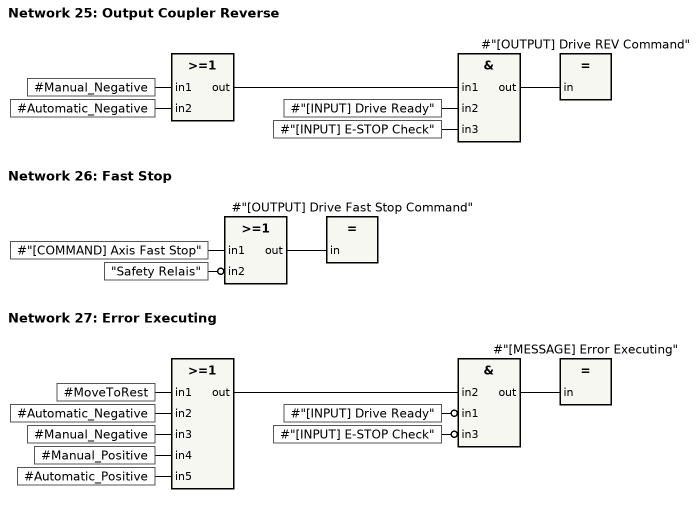
   #"[OUTPUT] Drive REV Command" := (#Manual_Negative OR #Automatic_Negative) AND #"[INPUT] Drive Ready" AND #"[INPUT] E-STOP Check";
END_REGION

REGION Network 26: Fast Stop
   #"[OUTPUT] Drive Fast Stop Command" := #"[COMMAND] Axis Fast Stop" OR NOT "Safety Relais";
END_REGION

REGION Network 27: Error Executing
   #"[MESSAGE] Error Executing" := (#MoveToRest OR #Automatic_Negative OR #Manual_Negative OR #Manual_Positive OR #Automatic_Positive) AND NOT #"[INPUT] Drive Ready" AND NOT #"[INPUT] E-STOP Check";
END_REGION
END_FUNCTION

FUNCTION "EncoderFeedback" : Void   // FC16, FBD
TITLE = EncoderFeedback Block
VERSION : 0.1
// stored: AutoNumber true, IsIECCheckEnabled false, UDAEnableTagReadback false
   VAR_INPUT
      CounterTag : Int;   // Connect to the CounterTag IW102
      Position_Offset : Real;   // Fill in the tolerance, when the axis approves the position. Above or below the desired position
      Pulsfactor : Real;   // Number of pulses after 360 degree turn of the axis.
      Position_Correction : Real;   // Small Position Correction for the Axis
      ReferenceRun_Command : Bool;   // Command of starting the referencerun
      ReferenceSwitch : Bool;   // ReferenceSwitch Mounted on Axis
      ReferencePosition : Int;   // Position where the index puls of the reference switch enters.
   END_VAR
   VAR_OUTPUT
      Scaled_Position : Real;   // Scaled Position scaled with Pulsfactor
      Actual_Enc_Pos : Real;   // Actual Encoder Position
      AxisDB_Connection : Real;   // Connection with Axis DB connection
   END_VAR
   VAR_TEMP
      Corrected_Axis_Pos : Real;
      Unscaled_Position : Int;   // Unscaled Position of the Encoder
      Unsc2 : Int;   // Unsc 2 position
      Act_Enc_Pos_Int : DInt;
      Scaled_Position_Real : Real;
      PosDint : DInt;
      Unscaled_Position_Real : Real;
      InternalCounter : Int;
      CalDifCounter : Int;
      Pos_Storage : Int;
      Pos_Diffrence : Int;
      Add_Pos : Int;
      Sub_Pos : Int;
      LessThanZero : Bool;
      LTZ_out : Int;
   END_VAR
BEGIN

REGION Network 1: SPARE
END_REGION

NETWORK
TITLE = Call the Countermodule
      L     #CounterTag;  //Van tellerkaart TAG Gelinkt aan IW102
      L     "PositionManagement".Data.CntPlsPrev;  //Vorige scan
      -D;
      T     "PositionManagement".Data.CntPlsDiff;  //Verschil

      L     "PositionManagement".Data.CntPlsDiff;  // Verschil groter dan nul?
      L     0;
      >D;
      JCN   chkneg;

      L     "PositionManagement".Data.CntPlsDiff;  //Verschil optellen bij actuele pulswaarde
      L     "PositionManagement".Data.CntPlsAct;
      +D;
      T     "PositionManagement".Data.CntPlsAct;
      JU    end;  //rest overslaan.

chkneg:L     "PositionManagement".Data.CntPlsDiff;  // Verschil groter dan nul?
      L     0;
      <D;
      JCN   end;
      L     -1;  //verschil positief maken
      *D;
      T     "PositionManagement".Data.CntPlsDiff;  //verschil positief

      L     "PositionManagement".Data.CntPlsAct;  //Verschil optellen bij actuele pulswaarde
      +D;
      T     "PositionManagement".Data.CntPlsAct;

end:  NOP   0;

      L     #CounterTag;
      T     "PositionManagement".Data.CntPlsPrev;


REGION Network 3: Store Old Position
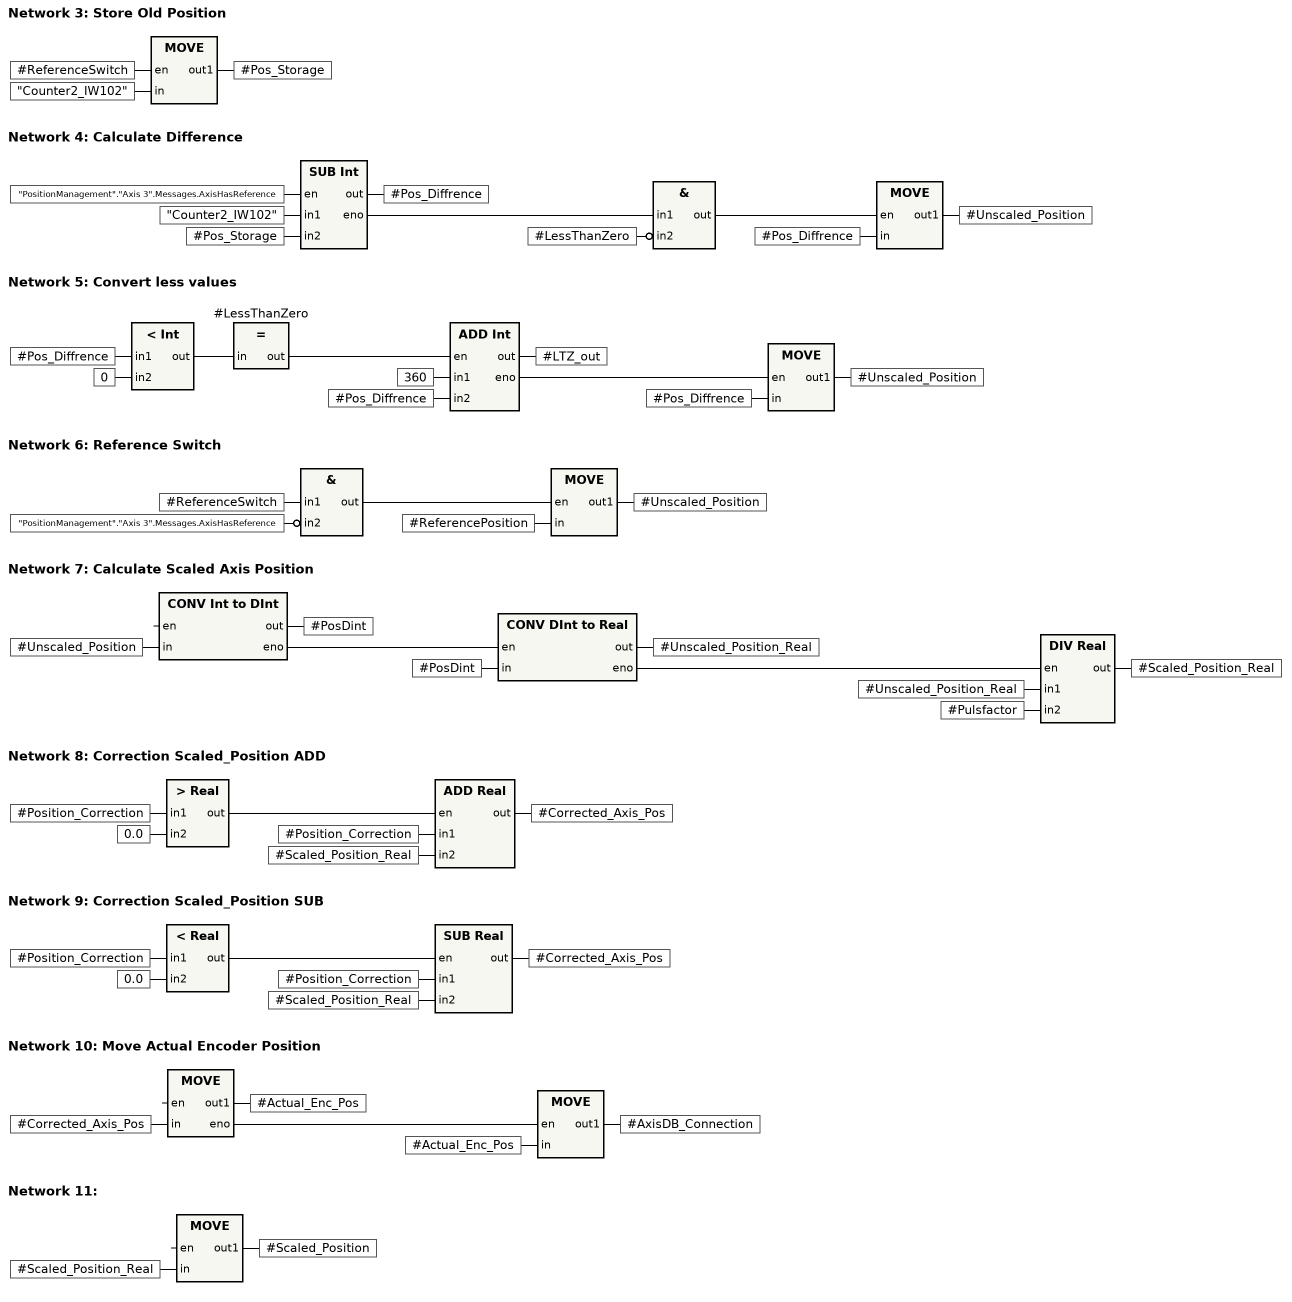
   IF #ReferenceSwitch THEN #Pos_Storage := "Counter2_IW102"; END_IF;
END_REGION

REGION Network 4: Calculate Difference
   // ENO of a box is taken as its EN; it also drops when the box reports an error
   IF "PositionManagement"."Axis 3".Messages.AxisHasReference THEN
       #Pos_Diffrence := "Counter2_IW102" - #Pos_Storage;
   END_IF;
   IF "PositionManagement"."Axis 3".Messages.AxisHasReference AND NOT #LessThanZero THEN
       #Unscaled_Position := #Pos_Diffrence;
   END_IF;
END_REGION

REGION Network 5: Convert less values
   // ENO of a box is taken as its EN; it also drops when the box reports an error
   #LessThanZero := #Pos_Diffrence < 0;
   IF #LessThanZero THEN
       #LTZ_out := 360 + #Pos_Diffrence;
       #Unscaled_Position := #Pos_Diffrence;
   END_IF;
END_REGION

REGION Network 6: Reference Switch
   IF #ReferenceSwitch AND NOT "PositionManagement"."Axis 3".Messages.AxisHasReference THEN
       #Unscaled_Position := #ReferencePosition;
   END_IF;
END_REGION

REGION Network 7: Calculate Scaled Axis Position
   // ENO of a box is taken as its EN; it also drops when the box reports an error
   #PosDint := INT_TO_DINT(#Unscaled_Position);
   #Unscaled_Position_Real := DINT_TO_REAL(#PosDint);
   #Scaled_Position_Real := #Unscaled_Position_Real / #Pulsfactor;
END_REGION

REGION Network 8: Correction Scaled_Position ADD
   IF #Position_Correction > 0.0 THEN
       #Corrected_Axis_Pos := #Position_Correction + #Scaled_Position_Real;
   END_IF;
END_REGION

REGION Network 9: Correction Scaled_Position SUB
   IF #Position_Correction < 0.0 THEN
       #Corrected_Axis_Pos := #Position_Correction - #Scaled_Position_Real;
   END_IF;
END_REGION

REGION Network 10: Move Actual Encoder Position
   // ENO of a box is taken as its EN; it also drops when the box reports an error
   #Actual_Enc_Pos := #Corrected_Axis_Pos;
   #AxisDB_Connection := #Actual_Enc_Pos;
END_REGION

REGION Network 11
   #Scaled_Position := #Scaled_Position_Real;
END_REGION
END_FUNCTION

FUNCTION_BLOCK "MC_Move"   // FB10, FBD
TITLE = MC_Move
VERSION : 0.1
// Block moves an Axis to an Desired Position, this block comes with the brake feature. When the axis is on position it keeps the brake for a time. You can set the time in the Brake Time field.
// stored: AutoNumber true, IsIECCheckEnabled false, UDAEnableTagReadback false
   VAR_INPUT
      Start : Bool;
      "Desired Position" : Real;
      "Speed (50-75%)" : Int;
      "Brake on Position" : Bool;
      Acceleration : Real;
      Deacceleration : Real;
      "Drive Ready" : Bool;
      "Drive On Position" : Bool;
      "Brake Time" : Time := T#500ms;
      "Safety OK" : Bool;
   END_VAR
   VAR_OUTPUT
      Go : Bool;
      "Desired Position Out" : Real;
      "Speed Output" : Int;
      "Acceleration Out" : Real;
      "Deacceleration Out" : Real;
      "Brake Out" : Bool;
   END_VAR
   VAR_TEMP
      SR_1 : Bool;
   END_VAR
BEGIN

REGION Network 1: Start - Go To Position + Speed
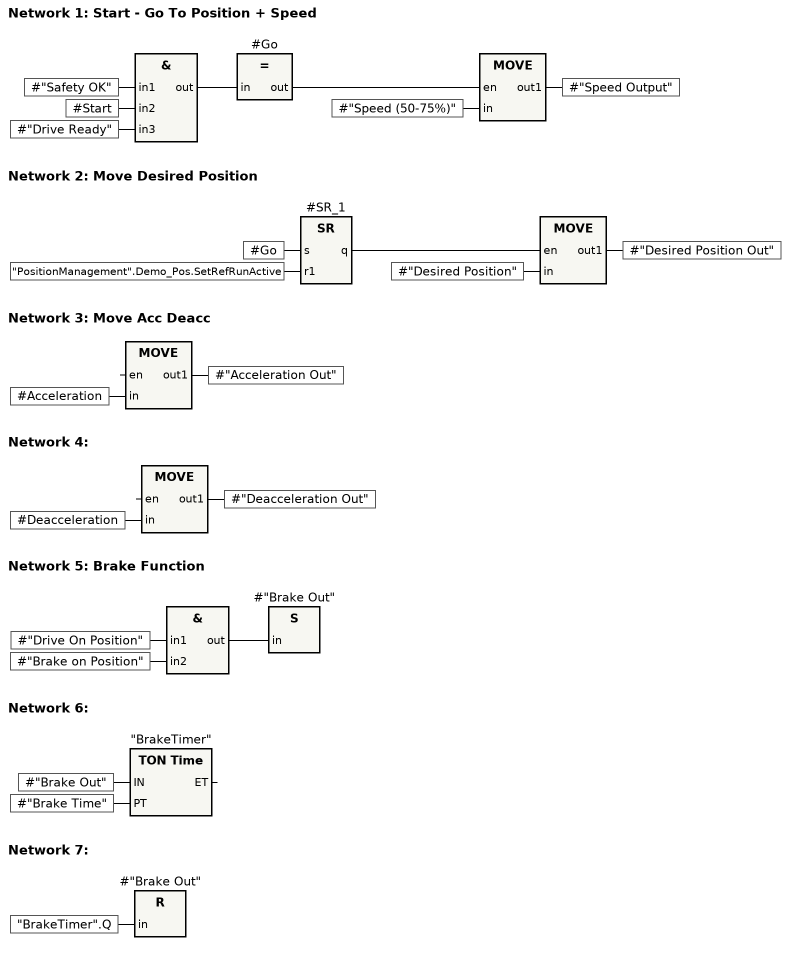
   #Go := #"Safety OK" AND #Start AND #"Drive Ready";
   IF #Go THEN #"Speed Output" := #"Speed (50-75%)"; END_IF;
END_REGION

REGION Network 2: Move Desired Position
   IF #Go THEN
       #SR_1 := TRUE;   // SR flip-flop
   END_IF;
   IF "PositionManagement".Demo_Pos.SetRefRunActive THEN #SR_1 := FALSE; END_IF;
   IF #SR_1 THEN #"Desired Position Out" := #"Desired Position"; END_IF;
END_REGION

REGION Network 3: Move Acc Deacc
   #"Acceleration Out" := #Acceleration;
END_REGION

REGION Network 4
   #"Deacceleration Out" := #Deacceleration;
END_REGION

REGION Network 5: Brake Function
   IF #"Drive On Position" AND #"Brake on Position" THEN #"Brake Out" := TRUE; END_IF;
END_REGION

REGION Network 6
   "BrakeTimer".TON(IN := #"Brake Out", PT := #"Brake Time");
END_REGION

REGION Network 7
   IF "BrakeTimer".Q THEN #"Brake Out" := FALSE; END_IF;
END_REGION
END_FUNCTION_BLOCK

FUNCTION_BLOCK "MC_Jog"   // FB11, FBD
TITLE = MC_Jog
VERSION : 0.1
// With this block you can Jog an Axis manual, you can set the speed on 25%, 50% or 75%. It also has an brake functionality, when you set Brake to true, it holds the brake for 2 seconds, then releases it.
// stored: AutoNumber true, IsIECCheckEnabled false, UDAEnableTagReadback false
   VAR_INPUT
      "Jog Forward" : Bool;
      "Jog Backward" : Bool;
      Speed : Int;
      Brake : Bool;
   END_VAR
   VAR_OUTPUT
      "Drive Fwd Output" : Bool;
      "Drive Rev Output" : Bool;
      "Drive Speed Output" : Int;
      "Drive Brake Output" : Bool;
   END_VAR
BEGIN

REGION Network 1: Manual Control
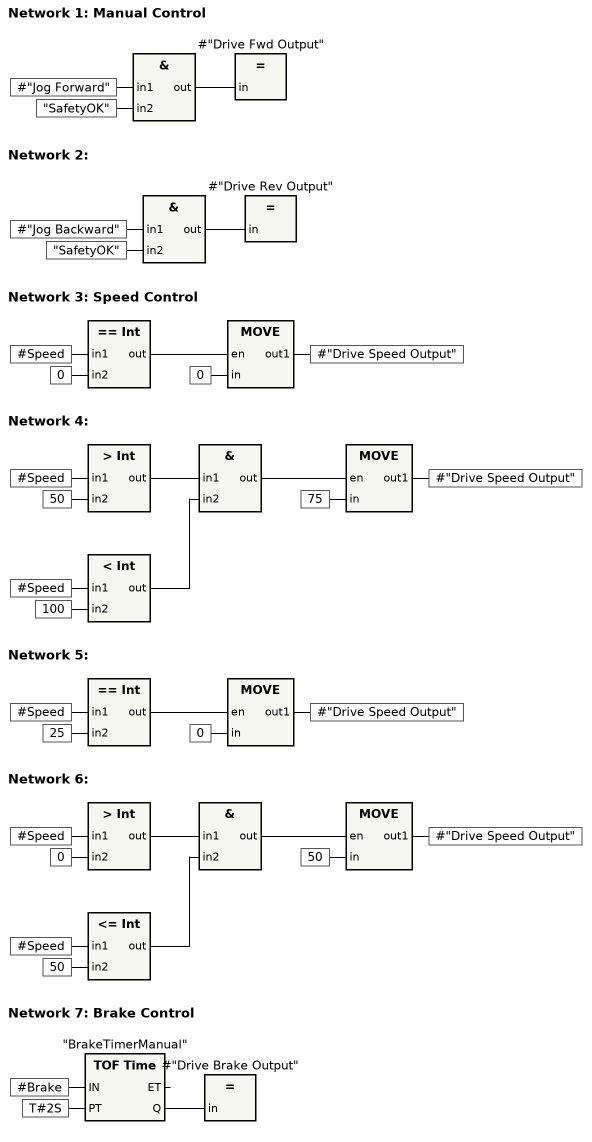
   #"Drive Fwd Output" := #"Jog Forward" AND "SafetyOK";
END_REGION

REGION Network 2
   #"Drive Rev Output" := #"Jog Backward" AND "SafetyOK";
END_REGION

REGION Network 3: Speed Control
   IF #Speed = 0 THEN #"Drive Speed Output" := 0; END_IF;
END_REGION

REGION Network 4
   IF (#Speed > 50) AND (#Speed < 100) THEN #"Drive Speed Output" := 75; END_IF;
END_REGION

REGION Network 5
   IF #Speed = 25 THEN #"Drive Speed Output" := 0; END_IF;
END_REGION

REGION Network 6
   IF (#Speed > 0) AND (#Speed <= 50) THEN #"Drive Speed Output" := 50; END_IF;
END_REGION

REGION Network 7: Brake Control
   "BrakeTimerManual".TOF(IN := #Brake, PT := T#2S);
   #"Drive Brake Output" := "BrakeTimerManual".Q;
END_REGION
END_FUNCTION_BLOCK

FUNCTION_BLOCK "ProductBuffer_V3"
{ S7_Optimized_Access := 'FALSE' }
VERSION : 0.1
   VAR_INPUT 
      SensorInput : Bool;   // Sensor aan begin band
      EncoderPosition : Real;   // Koppel aan Encoder Data Instance
      TriggerDistance : Real;   // Gewenste Afstand Product voor trigger
      TriggerFeedback : Bool;
   END_VAR

   VAR_OUTPUT 
      TriggerMovement : Bool;   // Trigger Start Movement
      ProductCount : Int;   // Count products in buffer
   END_VAR

   VAR 
      ProductBuffer { S7_SetPoint := 'False'} : Array[0..9] of "ProductTrack";
      PrevSensor { S7_SetPoint := 'True'} : Bool;
      MovementActive : Bool;
      i : Int;
      Distance : Real;
   END_VAR


BEGIN
	// 1️⃣ Flankdetectie - detecteer nieuw product
	IF #SensorInput AND NOT #PrevSensor THEN
	    FOR #i := 0 TO 9 DO
	        IF NOT #ProductBuffer[#i].Active THEN
	            #ProductBuffer[#i].StartPosition := #EncoderPosition;
	            #ProductBuffer[#i].Active := TRUE;
	            EXIT;
	        END_IF;
	    END_FOR;
	END_IF;
	#PrevSensor := #SensorInput;
	
	// 2️⃣ Tel actieve producten
	#ProductCount := 0;
	FOR #i := 0 TO 9 DO
	    IF #ProductBuffer[#i].Active THEN
	        #ProductCount := #ProductCount + 1;
	    END_IF;
	END_FOR;
	
	// 3️⃣ Zoek eerste product dat zijn afstand heeft afgelegd
	IF NOT #MovementActive THEN
	    FOR #i := 0 TO 9 DO
	        IF #ProductBuffer[#i].Active THEN
	            #Distance := #EncoderPosition - #ProductBuffer[#i].StartPosition;
	            
	            IF #Distance >= #TriggerDistance THEN
	                #TriggerMovement := TRUE;
	                #MovementActive := TRUE;
	                #ProductBuffer[#i].Active := FALSE;
	                EXIT;
	            END_IF;
	        END_IF;
	    END_FOR;
	END_IF;
	
	// 4️⃣ Wacht op feedback om beweging af te ronden
	IF #MovementActive AND #TriggerFeedback THEN
	    #TriggerMovement := FALSE;
	    #MovementActive := FALSE;
	END_IF;
	
END_FUNCTION_BLOCK

FUNCTION_BLOCK "Programma 1 - Test"   // FB12, GRAPH
VERSION : 0.1
// stored: AcknowledgeErrorsRequired true, AutoNumber true, CreateMinimizedDB false, IsIECCheckEnabled false, LanguageInNetworks LAD, LockOperatingMode false, PermanentILProcessingInMANMode false, SkipSteps false, UDAEnableTagReadback false, WithAlarmHandling true
   VAR_INPUT
      OFF_SQ { ExternalAccessible := 'False'; ExternalVisible := 'False'; ExternalWritable := 'False'} : Bool := false;   // Turn sequence off
      INIT_SQ { ExternalAccessible := 'False'; ExternalVisible := 'False'; ExternalWritable := 'False'} : Bool := false;   // Set sequence to initial state
      ACK_EF { ExternalAccessible := 'False'; ExternalVisible := 'False'; ExternalWritable := 'False'} : Bool := false;   // Acknowledge all errors and faults
      S_PREV { ExternalAccessible := 'False'; ExternalVisible := 'False'; ExternalWritable := 'False'} : Bool := false;   // Output previous step in parameter S_NO
      S_NEXT { ExternalAccessible := 'False'; ExternalVisible := 'False'; ExternalWritable := 'False'} : Bool := false;   // Indicate next step in parameter S_NO
      SW_AUTO { ExternalAccessible := 'False'; ExternalVisible := 'False'; ExternalWritable := 'False'} : Bool := false;   // Automatic mode
      SW_TAP { ExternalAccessible := 'False'; ExternalVisible := 'False'; ExternalWritable := 'False'} : Bool := false;   // Semiautomatic/switch with transition
      SW_TOP { ExternalAccessible := 'False'; ExternalVisible := 'False'; ExternalWritable := 'False'} : Bool := false;   // Semiautomatic/ignore transition
      SW_MAN { ExternalAccessible := 'False'; ExternalVisible := 'False'; ExternalWritable := 'False'} : Bool := false;   // Manual mode
      S_SEL { ExternalAccessible := 'False'; ExternalVisible := 'False'; ExternalWritable := 'False'} : Int := 0;   // Select step to be output to S_NO
      S_ON { ExternalAccessible := 'False'; ExternalVisible := 'False'; ExternalWritable := 'False'} : Bool := false;   // Activate step indicated in S_NO
      S_OFF { ExternalAccessible := 'False'; ExternalVisible := 'False'; ExternalWritable := 'False'} : Bool := false;   // Deactivate step indicated S_NO
      T_PUSH { ExternalAccessible := 'False'; ExternalVisible := 'False'; ExternalWritable := 'False'} : Bool := false;   // Enable transition to switch in semi automatic mode
      "Confimation Position 1" : Bool;
      "Confirmation Position 2" : Bool;
      "Products more than zero" : Bool;
      "Products zero" : Bool;
      "Timer 1" : Time;
   END_VAR
   VAR_OUTPUT
      S_NO { ExternalAccessible := 'False'; ExternalVisible := 'False'; ExternalWritable := 'False'} : Int := 0;   // Step number
      S_MORE { ExternalAccessible := 'False'; ExternalVisible := 'False'; ExternalWritable := 'False'} : Bool := false;   // More steps are available and can be shown in S_NO
      S_ACTIVE { ExternalAccessible := 'False'; ExternalVisible := 'False'; ExternalWritable := 'False'} : Bool := false;   // Step indicated in S_NO is active
      ERR_FLT { ExternalAccessible := 'False'; ExternalVisible := 'False'; ExternalWritable := 'False'} : Bool := false;   // Interlock or supervision group error
      AUTO_ON { ExternalAccessible := 'False'; ExternalVisible := 'False'; ExternalWritable := 'False'} : Bool := false;   // Automatic mode is active
      TAP_ON { ExternalAccessible := 'False'; ExternalVisible := 'False'; ExternalWritable := 'False'} : Bool := false;   // Semiautomatic mode/step with transition enabled
      TOP_ON { ExternalAccessible := 'False'; ExternalVisible := 'False'; ExternalWritable := 'False'} : Bool := false;   // Semiautomatic mode/ignore transition enabled
      MAN_ON { ExternalAccessible := 'False'; ExternalVisible := 'False'; ExternalWritable := 'False'} : Bool := false;   // Manual mode is active
      "Move Position 1" : Bool;
      "Move Position 2" : Bool;
   END_VAR
   VAR DB_SPECIFIC
      S_DISPLAY { ExternalAccessible := 'False'; ExternalVisible := 'False'; ExternalWritable := 'False'} : Int;   // Internal display of output parameter S_NO
      S_SEL_OLD { ExternalAccessible := 'False'; ExternalVisible := 'False'; ExternalWritable := 'False'} : Int;   // Previous value in S_SEL
      S_DISPIDX { ExternalAccessible := 'False'; ExternalVisible := 'False'; ExternalWritable := 'False'} : Byte;   // Index of the step in S_NO
      T_DISPIDX { ExternalAccessible := 'False'; ExternalVisible := 'False'; ExternalWritable := 'False'} : Byte;   // Index of the transition displayed in T_NO
      MOP { ExternalAccessible := 'False'; ExternalVisible := 'False'; ExternalWritable := 'False'} : Struct   // Mode
         AUTO { ExternalAccessible := 'False'; ExternalVisible := 'False'; ExternalWritable := 'False'} : Bool := true;   // Status: automatic mode
         MAN { ExternalAccessible := 'False'; ExternalVisible := 'False'; ExternalWritable := 'False'} : Bool := false;   // Status: manual mode
         TAP { ExternalAccessible := 'False'; ExternalVisible := 'False'; ExternalWritable := 'False'} : Bool := false;   // Status: semi automatic/switch with transition
         TOP { ExternalAccessible := 'False'; ExternalVisible := 'False'; ExternalWritable := 'False'} : Bool := false;   // Status: semi automatic/ignore transition
         ACK_S { ExternalAccessible := 'False'; ExternalVisible := 'False'; ExternalWritable := 'False'} : Bool := false;   // Request: acknowledge step at parameter S_NO
         REG_S { ExternalAccessible := 'False'; ExternalVisible := 'False'; ExternalWritable := 'False'} : Bool := false;   // Request: register step indicated in S_NO
         T_PREV { ExternalAccessible := 'False'; ExternalVisible := 'False'; ExternalWritable := 'False'} : Bool := false;   // Request: output previous valid transition in T_NO
         T_NEXT { ExternalAccessible := 'False'; ExternalVisible := 'False'; ExternalWritable := 'False'} : Bool := false;   // Request: output next valid transition in T_NO
         LOCK { ExternalAccessible := 'False'; ExternalVisible := 'False'; ExternalWritable := 'False'} : Bool := true;   // Status: interlocks activated
         SUP { ExternalAccessible := 'False'; ExternalVisible := 'False'; ExternalWritable := 'False'} : Bool := true;   // Status: supervisions activated
         ACKREQ { ExternalAccessible := 'False'; ExternalVisible := 'False'; ExternalWritable := 'False'} : Bool := true;   // Status: acknowledgment required
         SSKIP { ExternalAccessible := 'False'; ExternalVisible := 'False'; ExternalWritable := 'False'} : Bool := false;   // Status: "Skip steps" enabled
         OFF { ExternalAccessible := 'False'; ExternalVisible := 'False'; ExternalWritable := 'False'} : Bool := false;   // Request: deactivate all steps
         INIT { ExternalAccessible := 'False'; ExternalVisible := 'False'; ExternalWritable := 'False'} : Bool := true;   // Request: set sequence to initial state
         HALT { ExternalAccessible := 'False'; ExternalVisible := 'False'; ExternalWritable := 'False'} : Bool := false;   // Status: sequence halted
         TMS_HALT { ExternalAccessible := 'False'; ExternalVisible := 'False'; ExternalWritable := 'False'} : Bool := false;   // Status: all internal timers held
         OPS_ZERO { ExternalAccessible := 'False'; ExternalVisible := 'False'; ExternalWritable := 'False'} : Bool := false;   // Status: set all operands processed with N, L, D instructions to 0
         SACT_DISP { ExternalAccessible := 'False'; ExternalVisible := 'False'; ExternalWritable := 'False'} : Bool := true;   // Status: display active steps only
         SEF_DISP { ExternalAccessible := 'False'; ExternalVisible := 'False'; ExternalWritable := 'False'} : Bool := false;   // Status: display only steps with errors and disrupted steps
         SALL_DISP { ExternalAccessible := 'False'; ExternalVisible := 'False'; ExternalWritable := 'False'} : Bool := false;   // Status: display all steps
         S_PREV { ExternalAccessible := 'False'; ExternalVisible := 'False'; ExternalWritable := 'False'} : Bool := false;   // Request: output previous step to S_NO
         S_NEXT { ExternalAccessible := 'False'; ExternalVisible := 'False'; ExternalWritable := 'False'} : Bool := false;   // Request: Output next step at S_NO parameter
         S_SELOK { ExternalAccessible := 'False'; ExternalVisible := 'False'; ExternalWritable := 'False'} : Bool := false;   // Request: output step number from S_SEL to S_NO
         S_ON { ExternalAccessible := 'False'; ExternalVisible := 'False'; ExternalWritable := 'False'} : Bool := false;   // Request: activate step indicated in S_NO
         S_OFF { ExternalAccessible := 'False'; ExternalVisible := 'False'; ExternalWritable := 'False'} : Bool := false;   // Request: deactivate step at parameter S_NO
         T_PUSH { ExternalAccessible := 'False'; ExternalVisible := 'False'; ExternalWritable := 'False'} : Bool := false;   // Request: transition switching enabled
         REG { ExternalAccessible := 'False'; ExternalVisible := 'False'; ExternalWritable := 'False'} : Bool := false;   // Request: register all interlock and supervision errors
         ACK { ExternalAccessible := 'False'; ExternalVisible := 'False'; ExternalWritable := 'False'} : Bool := false;   // Request: acknowledge all interlock and supervision errors
         IL_PERM { ExternalAccessible := 'False'; ExternalVisible := 'False'; ExternalWritable := 'False'} : Bool := false;   // Status: permanent processing of all interlocks
         T_PERM { ExternalAccessible := 'False'; ExternalVisible := 'False'; ExternalWritable := 'False'} : Bool := false;   // Status: permanent processing of all transitions
         ILP_MAN { ExternalAccessible := 'False'; ExternalVisible := 'False'; ExternalWritable := 'False'} : Bool := false;   // Status: permanent processing of all interlocks in manual mode
      END_STRUCT;
      TICKS { ExternalAccessible := 'False'; ExternalVisible := 'False'; ExternalWritable := 'False'} : Struct   // Clock speeds
         DELTA { ExternalAccessible := 'False'; ExternalVisible := 'False'; ExternalWritable := 'False'} : Time := T#0ms;   // Time difference between cycles
         OLD { ExternalAccessible := 'False'; ExternalVisible := 'False'; ExternalWritable := 'False'} : Time := T#0ms;   // 10 ms clock counter value in last cycle
         NEW { ExternalAccessible := 'False'; ExternalVisible := 'False'; ExternalWritable := 'False'} : Time := T#0ms;   // 10 ms clock counter value in this cycle
      END_STRUCT;
      SQ_FLAGS { ExternalAccessible := 'False'; ExternalVisible := 'False'; ExternalWritable := 'False'} : Struct   // Sequence bit memory
         ERR_FLT { ExternalAccessible := 'False'; ExternalVisible := 'False'; ExternalWritable := 'False'} : Bool := false;   // Interlock and supervision group error
         ERROR { ExternalAccessible := 'False'; ExternalVisible := 'False'; ExternalWritable := 'False'} : Bool := false;   // Interlock group error
         FAULT { ExternalAccessible := 'False'; ExternalVisible := 'False'; ExternalWritable := 'False'} : Bool := false;   // Supervision group error
         RT_FAIL { ExternalAccessible := 'False'; ExternalVisible := 'False'; ExternalWritable := 'False'} : Bool := false;   // Runtime error
         NO_SNO { ExternalAccessible := 'False'; ExternalVisible := 'False'; ExternalWritable := 'False'} : Bool := false;   // Requested step number not found
         NF_OFL { ExternalAccessible := 'False'; ExternalVisible := 'False'; ExternalWritable := 'False'} : Bool := false;   // Overflow: too many ON or OFF requests
         SA_OFL { ExternalAccessible := 'False'; ExternalVisible := 'False'; ExternalWritable := 'False'} : Bool := false;   // Overflow: too many steps active
         TV_OFL { ExternalAccessible := 'False'; ExternalVisible := 'False'; ExternalWritable := 'False'} : Bool := false;   // Overflow: too many valid transitions
         MSG_OFL { ExternalAccessible := 'False'; ExternalVisible := 'False'; ExternalWritable := 'False'} : Bool := false;   // Overflow: not enough system resources for ALARM_S
         NO_SWI { ExternalAccessible := 'False'; ExternalVisible := 'False'; ExternalWritable := 'False'} : Bool := false;   // Do not switch in this cycle
         CYC_OP { ExternalAccessible := 'False'; ExternalVisible := 'False'; ExternalWritable := 'False'} : Bool := false;   // Cyclic execution of the sequence after initialization
         AS_MSG { ExternalAccessible := 'False'; ExternalVisible := 'False'; ExternalWritable := 'False'} : Bool := true;   // Alarms during runtime enabled or disabled by instruction
         AS_SEND { ExternalAccessible := 'False'; ExternalVisible := 'False'; ExternalWritable := 'False'} : Bool := false;   // Send alarms from WR_USMSG or only enter in diagnostics buffer
         SQ_BUSY { ExternalAccessible := 'False'; ExternalVisible := 'False'; ExternalWritable := 'False'} : Bool := false;   // Internal edge memory bit for sequence processing
         SA_BUSY { ExternalAccessible := 'False'; ExternalVisible := 'False'; ExternalWritable := 'False'} : Bool := false;   // Internal edge memory bit for sequence processing
         AS_SIG { ExternalAccessible := 'False'; ExternalVisible := 'False'; ExternalWritable := 'False'} : Bool := false;   // Edge memory bit for alarms from Alarm_S and Alarm_SQ
      END_STRUCT;
   END_VAR
BEGIN
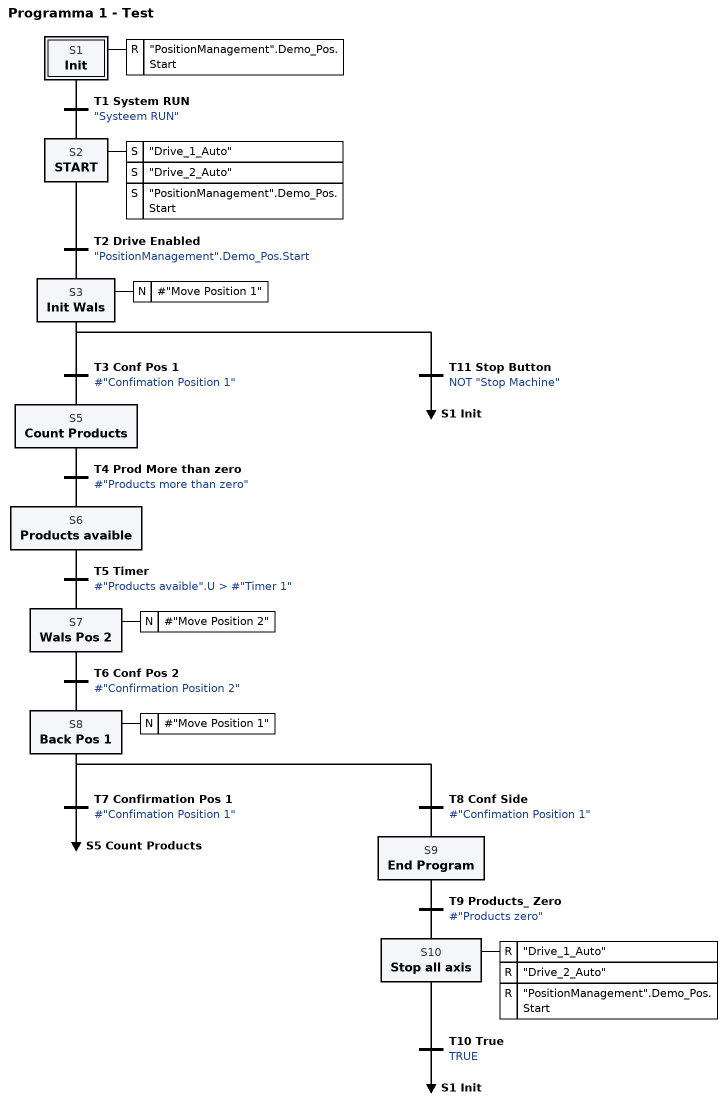
   // sequencer 1: SFC Program
   INITIAL_STEP Init:   // S1
              R    "PositionManagement".Demo_Pos.Start
   END_STEP
   TRANSITION "System RUN" FROM Init TO START   // T1
      := "Systeem RUN";
   END_TRANSITION
   STEP START:   // S2
      // Set Ouputs
              S    "Drive_1_Auto"
              S    "Drive_2_Auto"
              S    "PositionManagement".Demo_Pos.Start
   END_STEP
   TRANSITION "Drive Enabled" FROM START TO "Init Wals"   // T2
      := "PositionManagement".Demo_Pos.Start;
   END_TRANSITION
   STEP "Init Wals":   // S3
      // Move Start Position4
              N    #"Move Position 1"
   END_STEP
   TRANSITION "Conf Pos 1" FROM "Init Wals" TO "Count Products"   // T3
      := #"Confimation Position 1";
   END_TRANSITION
   TRANSITION "Stop Button" FROM "Init Wals" TO Init   // T11, jump
      := NOT "Stop Machine";
   END_TRANSITION
   STEP "Count Products":   // S5
   END_STEP
   TRANSITION "Prod More than zero" FROM "Count Products" TO "Products avaible"   // T4
      := #"Products more than zero";
   END_TRANSITION
   STEP "Products avaible":   // S6
   END_STEP
   TRANSITION "Timer" FROM "Products avaible" TO "Wals Pos 2"   // T5: Timer 1
      := #"Products avaible".U > #"Timer 1";
   END_TRANSITION
   STEP "Wals Pos 2":   // S7
              N    #"Move Position 2"
   END_STEP
   TRANSITION "Conf Pos 2" FROM "Wals Pos 2" TO "Back Pos 1"   // T6
      := #"Confirmation Position 2";
   END_TRANSITION
   STEP "Back Pos 1":   // S8
      // Move Position 1
              N    #"Move Position 1"
   END_STEP
   TRANSITION "Confirmation Pos 1" FROM "Back Pos 1" TO "Count Products"   // T7, jump: Conf Pos 1
      := #"Confimation Position 1";
   END_TRANSITION
   TRANSITION "Conf Side" FROM "Back Pos 1" TO "End Program"   // T8
      := #"Confimation Position 1";
   END_TRANSITION
   STEP "End Program":   // S9
   END_STEP
   TRANSITION "Products_ Zero" FROM "End Program" TO "Stop all axis"   // T9
      := #"Products zero";
   END_TRANSITION
   STEP "Stop all axis":   // S10
      // Reset Axis
              R    "Drive_1_Auto"
              R    "Drive_2_Auto"
              R    "PositionManagement".Demo_Pos.Start
   END_STEP
   TRANSITION True FROM "Stop all axis" TO Init   // T10, jump
      := TRUE;
   END_TRANSITION
END_FUNCTION_BLOCK

FUNCTION_BLOCK "Ouput_Function_1"   // FB8, FBD
TITLE = Ouput Controller Function Block
VERSION : 0.1
// stored: AutoNumber true, IsIECCheckEnabled false, UDAEnableTagReadback false
   VAR_INPUT
      "Stop Contact" : Bool;
      "Manual Command" : Bool;
      "Auto Command" : Bool;
      "Option Command" : Bool;
      "Disable Command" : Bool;
   END_VAR
   VAR_OUTPUT
      "Ouput Signal" : Bool;
   END_VAR
BEGIN

REGION Network 1: Ouput Controller
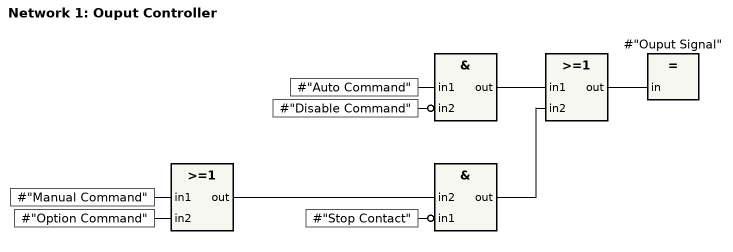
   #"Ouput Signal" := (#"Auto Command" AND NOT #"Disable Command") OR ((#"Manual Command" OR #"Option Command") AND NOT #"Stop Contact");
END_REGION
END_FUNCTION_BLOCK

FUNCTION_BLOCK "FB_EncoderFeedback_Degree"   // FB19, FBD
VERSION : 0.1
// stored: AutoNumber true, IsIECCheckEnabled false, UDAEnableTagReadback false
   VAR_INPUT
      CounterTag { ExternalVisible := 'False'; ExternalWritable := 'False'} : Int;   // Connect to the CounterTag IW102
      Position_Offset { ExternalVisible := 'False'; ExternalWritable := 'False'} : Real;   // Fill in the tolerance, when the axis approves the position. Above or below the desired position
      Pulsfactor { ExternalVisible := 'False'; ExternalWritable := 'False'} : Real;   // Number of pulses after 360 degree turn of the axis.
      Position_Correction { ExternalVisible := 'False'; ExternalWritable := 'False'} : Real;   // Small Position Correction for the Axis
      ReferenceRun_Command { ExternalVisible := 'False'; ExternalWritable := 'False'} : Bool;   // Command of starting the referencerun
      ReferenceSwitch { ExternalVisible := 'False'; ExternalWritable := 'False'} : Bool;   // ReferenceSwitch Mounted on Axis
      ReferencePosition { ExternalVisible := 'False'; ExternalWritable := 'False'} : Int;   // Position where the index puls of the reference switch enters.
   END_VAR
   VAR_OUTPUT
      Scaled_Position { ExternalVisible := 'False'; ExternalWritable := 'False'} : Real;   // Scaled Position scaled with Pulsfactor
      Actual_Enc_Pos { ExternalVisible := 'False'; ExternalWritable := 'False'} : Real;   // Actual Encoder Position
      AxisDB_Connection { ExternalVisible := 'False'; ExternalWritable := 'False'} : Real;   // Connection with Axis DB connection
   END_VAR
   VAR_TEMP
      Corrected_Axis_Pos : Real;
      Unscaled_Position : Int;   // Unscaled Position of the Encoder
      Unsc2 : Int;   // Unsc 2 position
      Act_Enc_Pos_Int : DInt;
      Scaled_Position_Real : Real;
      PosDint : DInt;
      Unscaled_Position_Real : Real;
      InternalCounter : Int;
      CalDifCounter : Int;
      Pos_Storage : Int;
      Pos_Diffrence : Int;
      Add_Pos : Int;
      Sub_Pos : Int;
      LessThanZero : Bool;
      LTZ_out : Int;
   END_VAR
BEGIN

REGION Network 2: SPARE
END_REGION

NETWORK
TITLE = Call the Countermodule
      L     #CounterTag;  //Van tellerkaart TAG Gelinkt aan IW102
      L     "PositionManagement".Data.CntPlsPrev;  //Vorige scan
      -D;
      T     "PositionManagement".Data.CntPlsDiff;  //Verschil

      L     "PositionManagement".Data.CntPlsDiff;  // Verschil groter dan nul?
      L     0;
      >D;
      JCN   chkneg;

      L     "PositionManagement".Data.CntPlsDiff;  //Verschil optellen bij actuele pulswaarde
      L     "PositionManagement".Data.CntPlsAct;
      +D;
      T     "PositionManagement".Data.CntPlsAct;
      JU    end;  //rest overslaan.

chkneg:L     "PositionManagement".Data.CntPlsDiff;  // Verschil groter dan nul?
      L     0;
      <D;
      JCN   end;
      L     -1;  //verschil positief maken
      *D;
      T     "PositionManagement".Data.CntPlsDiff;  //verschil positief

      L     "PositionManagement".Data.CntPlsAct;  //Verschil optellen bij actuele pulswaarde
      +D;
      T     "PositionManagement".Data.CntPlsAct;

end:  NOP   0;

      L     #CounterTag;
      T     "PositionManagement".Data.CntPlsPrev;


REGION Network 4: Store Old Position
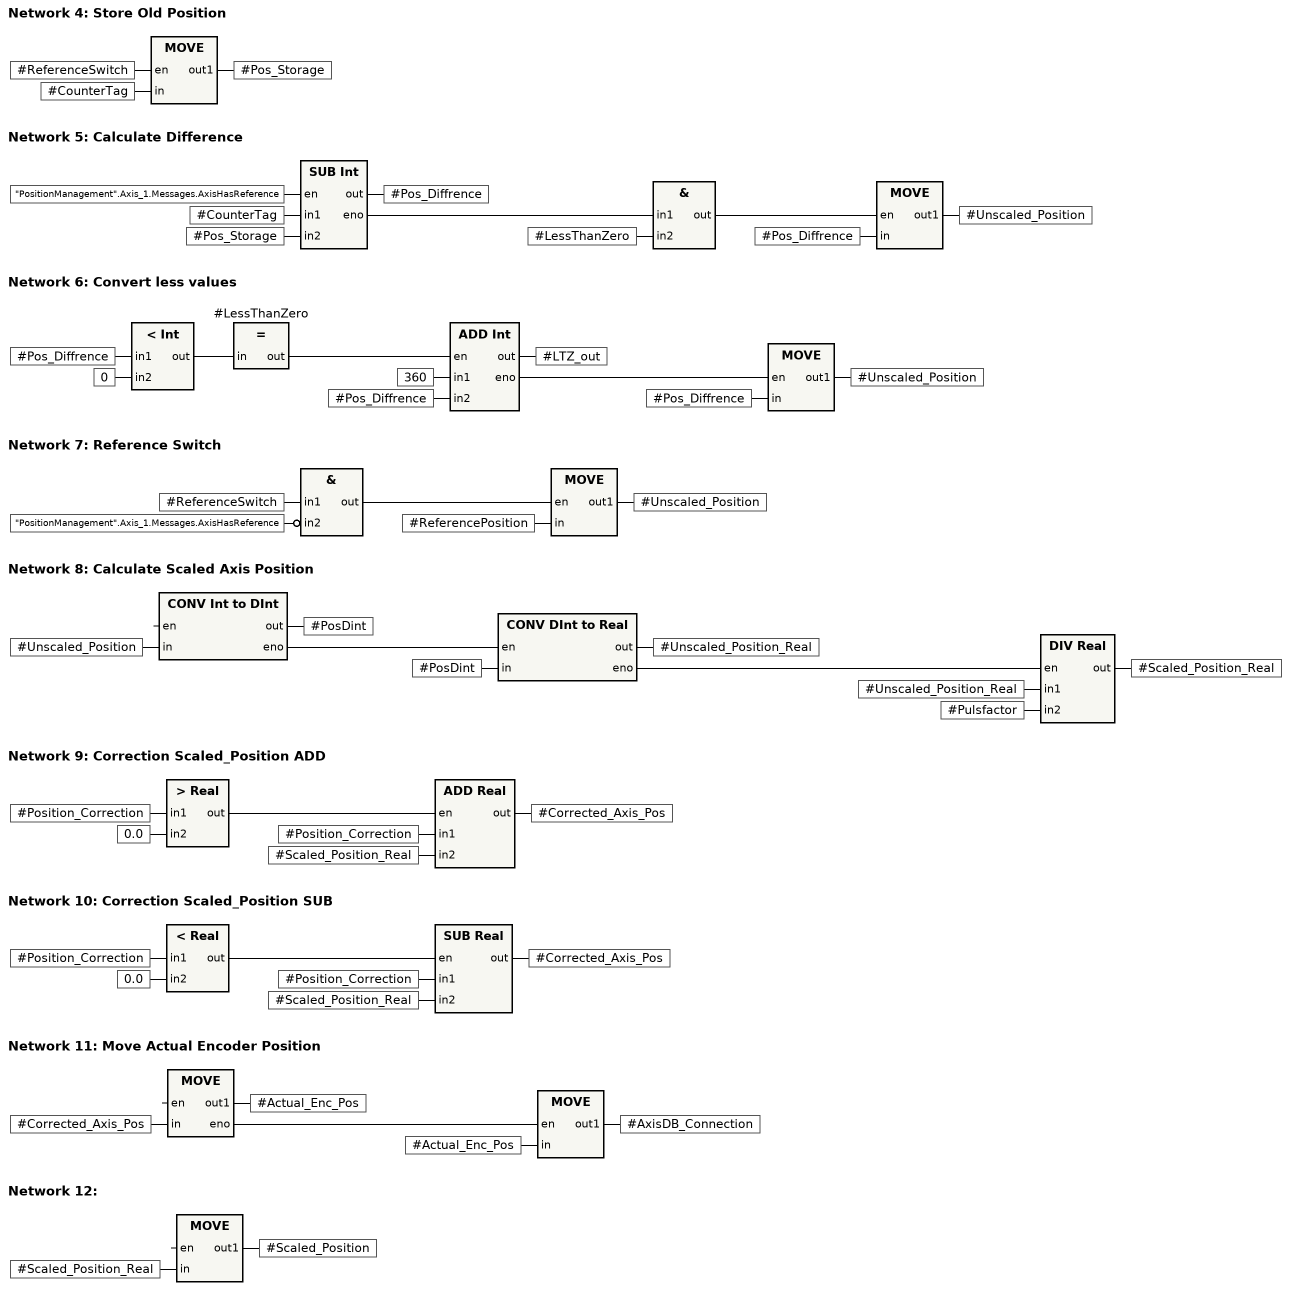
   IF #ReferenceSwitch THEN #Pos_Storage := #CounterTag; END_IF;
END_REGION

REGION Network 5: Calculate Difference
   // ENO of a box is taken as its EN; it also drops when the box reports an error
   IF "PositionManagement".Axis_1.Messages.AxisHasReference THEN
       #Pos_Diffrence := #CounterTag - #Pos_Storage;
   END_IF;
   IF "PositionManagement".Axis_1.Messages.AxisHasReference AND #LessThanZero THEN
       #Unscaled_Position := #Pos_Diffrence;
   END_IF;
END_REGION

REGION Network 6: Convert less values
   // ENO of a box is taken as its EN; it also drops when the box reports an error
   #LessThanZero := #Pos_Diffrence < 0;
   IF #LessThanZero THEN
       #LTZ_out := 360 + #Pos_Diffrence;
       #Unscaled_Position := #Pos_Diffrence;
   END_IF;
END_REGION

REGION Network 7: Reference Switch
   IF #ReferenceSwitch AND NOT "PositionManagement".Axis_1.Messages.AxisHasReference THEN
       #Unscaled_Position := #ReferencePosition;
   END_IF;
END_REGION

REGION Network 8: Calculate Scaled Axis Position
   // ENO of a box is taken as its EN; it also drops when the box reports an error
   #PosDint := INT_TO_DINT(#Unscaled_Position);
   #Unscaled_Position_Real := DINT_TO_REAL(#PosDint);
   #Scaled_Position_Real := #Unscaled_Position_Real / #Pulsfactor;
END_REGION

REGION Network 9: Correction Scaled_Position ADD
   IF #Position_Correction > 0.0 THEN
       #Corrected_Axis_Pos := #Position_Correction + #Scaled_Position_Real;
   END_IF;
END_REGION

REGION Network 10: Correction Scaled_Position SUB
   IF #Position_Correction < 0.0 THEN
       #Corrected_Axis_Pos := #Position_Correction - #Scaled_Position_Real;
   END_IF;
END_REGION

REGION Network 11: Move Actual Encoder Position
   // ENO of a box is taken as its EN; it also drops when the box reports an error
   #Actual_Enc_Pos := #Corrected_Axis_Pos;
   #AxisDB_Connection := #Actual_Enc_Pos;
END_REGION

REGION Network 12
   #Scaled_Position := #Scaled_Position_Real;
END_REGION
END_FUNCTION_BLOCK

DATA_BLOCK "BlowOff_Timer_Manual2DB"   // DB86
VERSION : 0.1
// stored: AutoNumber true, InstanceOfName BlowOff_Timer, InstanceOfType FB
"BlowOff_Timer"
   // VAR_INPUT
   //    Enable : Bool;
   //    CycleTime : Time;
   //    PulseDuration : Time;
   //    NowTime : Time;
   // END_VAR
   // VAR_OUTPUT
   //    Q_Pulse : Bool;
   // END_VAR
   // VAR RETAIN
   //    CycleTimer : TON;
   //    PulseTimer : TON;
   //    State { S7_SetPoint := 'True'} : Int;
   //    S_PEXT : Int;
   // END_VAR
BEGIN
END_DATA_BLOCK

DATA_BLOCK "BlowOff_Timer_ManualDB"   // DB83
VERSION : 0.1
// stored: AutoNumber true, InstanceOfName BlowOff_Timer, InstanceOfType FB
"BlowOff_Timer"
   // VAR_INPUT
   //    Enable : Bool;
   //    CycleTime : Time;
   //    PulseDuration : Time;
   //    NowTime : Time;
   // END_VAR
   // VAR_OUTPUT
   //    Q_Pulse : Bool;
   // END_VAR
   // VAR RETAIN
   //    CycleTimer : TON;
   //    PulseTimer : TON;
   //    State { S7_SetPoint := 'True'} : Int;
   //    S_PEXT : Int;
   // END_VAR
BEGIN
END_DATA_BLOCK

DATA_BLOCK "BlowOff_Timer_Prog1"   // DB75
VERSION : 0.1
// stored: AutoNumber true, InstanceOfName BlowOff_Timer, InstanceOfType FB
"BlowOff_Timer"
   // VAR_INPUT
   //    Enable : Bool;
   //    CycleTime : Time;
   //    PulseDuration : Time;
   //    NowTime : Time;
   // END_VAR
   // VAR_OUTPUT
   //    Q_Pulse : Bool;
   // END_VAR
   // VAR RETAIN
   //    CycleTimer : TON;
   //    PulseTimer : TON;
   //    State { S7_SetPoint := 'True'} : Int;
   //    S_PEXT : Int;
   // END_VAR
BEGIN
END_DATA_BLOCK

DATA_BLOCK "FB_EncoderFeedback_Aanvoerband"   // DB78
VERSION : 0.1
// stored: AutoNumber true, InstanceOfName FB_EncoderFeedback_Degree, InstanceOfType FB
"FB_EncoderFeedback_Degree"
BEGIN
END_DATA_BLOCK

DATA_BLOCK "FB_ProductTrigger_1"   // DB67
VERSION : 0.1
// stored: AutoNumber true, InstanceOfName FB_ProductTrigger, InstanceOfType FB
"FB_ProductTrigger"
   // VAR_INPUT
   //    SensorInput : Bool;
   //    TimeDelay : Time;
   //    SystemTime : Time;
   // END_VAR
   // VAR_OUTPUT
   //    TriggerMovement : Bool;
   //    ProductCount : Int;
   // END_VAR
BEGIN
END_DATA_BLOCK

DATA_BLOCK "FB_SystemTimeCounter_DB_1"   // DB23
VERSION : 0.1
// stored: AutoNumber true, InstanceOfName FB_SystemTimeCounter, InstanceOfType FB
"FB_SystemTimeCounter"
   // VAR_INPUT
   //    Enable : Bool;
   //    CycleTime : Time;
   // END_VAR
   // VAR_OUTPUT
   //    SystemTime : Time;
   // END_VAR
BEGIN
END_DATA_BLOCK

DATA_BLOCK "MC_Move_1"   // DB76
VERSION : 0.1
// stored: AutoNumber true, InstanceOfName MC_Move, InstanceOfType FB
"MC_Move"
BEGIN
END_DATA_BLOCK

DATA_BLOCK "MC_Move_DB"   // DB62
VERSION : 0.1
// stored: AutoNumber true, InstanceOfName MC_Move, InstanceOfType FB
"MC_Move"
BEGIN
END_DATA_BLOCK

DATA_BLOCK "MC_Move_Prog.1_1"   // DB59
VERSION : 0.1
// stored: AutoNumber true, InstanceOfName MC_Move, InstanceOfType FB
"MC_Move"
BEGIN
END_DATA_BLOCK

DATA_BLOCK "ProductBuffer_BehindWals"   // DB79
VERSION : 0.1
// stored: AutoNumber true, InstanceOfName ProductBuffer, InstanceOfType FB
"ProductBuffer"
   // VAR_INPUT
   //    SensorInput : Bool;
   //    TimeDelay : Time;
   //    TriggerFeedback : Bool;
   // END_VAR
   // VAR_OUTPUT
   //    TriggerMovement : Bool;
   //    ProductCount : Int;
   // END_VAR
   // VAR RETAIN
   //    PrevSensor : Bool;
   //    DelayTimer : TON;
   //    MovementActive { S7_SetPoint := 'True'} : Bool;
   // END_VAR
BEGIN
END_DATA_BLOCK

DATA_BLOCK "ProductBuffer_DB_Manual"   // DB85
VERSION : 0.1
// stored: AutoNumber true, InstanceOfName ProductBuffer, InstanceOfType FB
"ProductBuffer"
   // VAR_INPUT
   //    SensorInput : Bool;
   //    TimeDelay : Time;
   //    TriggerFeedback : Bool;
   // END_VAR
   // VAR_OUTPUT
   //    TriggerMovement : Bool;
   //    ProductCount : Int;
   // END_VAR
   // VAR RETAIN
   //    PrevSensor : Bool;
   //    DelayTimer : TON;
   //    MovementActive { S7_SetPoint := 'True'} : Bool;
   // END_VAR
BEGIN
END_DATA_BLOCK

DATA_BLOCK "ProductBuffer_V2_DB_BehindWals"   // DB82
VERSION : 0.1
// stored: AutoNumber true, InstanceOfName ProductBuffer_V2, InstanceOfType FB
"ProductBuffer_V2"
   // VAR_INPUT
   //    SensorInput : Bool;
   //    SensorManual : Bool;
   //    TimeDelay : Time;
   //    SystemTime : Time;
   //    TriggerFeedback : Bool;
   // END_VAR
   // VAR_OUTPUT
   //    TriggerMovement : Bool;
   //    InsertIndex { ExternalVisible := 'False'; ExternalWritable := 'False'} : Int;
   //    ProductCount : Int;
   //    SystemTicks : DInt;
   // END_VAR
   // VAR RETAIN
   //    ProductQueue : Array[0..1] of "ProductEntry";
   //    StartTimes : Struct
   //       _0 : Time;
   //       _1 : Time;
   //       _2 : Time;
   //       _3 : Time;
   //       _4 : Time;
   //       _5 : Time;
   //       _6 : Time;
   //       _7 : Time;
   //       _8 : Time;
   //       _9 : Time;
   //    END_STRUCT;
   //    Actives : Struct
   //       _0 : Bool;
   //       _1 : Bool;
   //       _2 : Bool;
   //       _3 : Bool;
   //       _4 : Bool;
   //       _5 : Bool;
   //       _6 : Bool;
   //       _7 : Bool;
   //       _8 : Bool;
   //       _9 : Bool;
   //    END_STRUCT;
   //    PrevSensor { ExternalVisible := 'False'; ExternalWritable := 'False'} : Bool;
   //    MovementActive { ExternalVisible := 'False'; ExternalWritable := 'False'} : Bool;
   //    i { ExternalVisible := 'False'; ExternalWritable := 'False'} : Int;
   //    Elapsed { ExternalVisible := 'False'; ExternalWritable := 'False'} : DInt;
   // END_VAR
BEGIN
END_DATA_BLOCK

DATA_BLOCK "ResetOuputs_Function_Rest"   // DB29
VERSION : 0.1
// stored: AutoNumber true, InstanceOfName ResetOuputs_Function, InstanceOfType FB
"ResetOuputs_Function"
BEGIN
END_DATA_BLOCK

DATA_BLOCK "FB_SystemTimeCounter_DB"   // DB69
VERSION : 0.1
// stored: AutoNumber true, InstanceOfName FB_SystemTimeCounter, InstanceOfType FB
"FB_SystemTimeCounter"
   // VAR_INPUT
   //    Enable : Bool;
   //    CycleTime : Time;
   // END_VAR
   // VAR_OUTPUT
   //    SystemTime : Time;
   // END_VAR
BEGIN
END_DATA_BLOCK

DATA_BLOCK "2in-1out_Block_LED-Estop"   // DB1
VERSION : 0.1
// stored: AutoNumber true, InstanceOfName 2in-1out_Block, InstanceOfType FB
"2in-1out_Block"
   // VAR_INPUT
   //    "Input Contact 1" : Bool;
   //    "Input Contact 2" : Bool;
   // END_VAR
   // VAR_OUTPUT
   //    "Output Contact 1" : Bool;
   // END_VAR
BEGIN
END_DATA_BLOCK

DATA_BLOCK "Alarm_Axis_Position_Function_Wals"   // DB41
VERSION : 0.1
// stored: AutoNumber true, InstanceOfName Alarm_Axis_Position_Function, InstanceOfType FB
"Alarm_Axis_Position_Function"
BEGIN
END_DATA_BLOCK

DATA_BLOCK "Alarm_Axis_Position_Function_Wals1"   // DB42
VERSION : 0.1
// stored: AutoNumber true, InstanceOfName Alarm_Axis_Position_Function, InstanceOfType FB
"Alarm_Axis_Position_Function"
BEGIN
END_DATA_BLOCK

DATA_BLOCK "DriveConfirmation_Function_Axis 3"   // DB47
VERSION : 0.1
// stored: AutoNumber true, InstanceOfName DriveConfirmation_Function, InstanceOfType FB
"DriveConfirmation_Function"
   // VAR_INPUT
   //    "System RUN" : Bool;
   //    "Drive Ouput Q" : Bool;
   //    "Drive Ready Signal" : Bool;
   //    DelayTime : Time;
   // END_VAR
   // VAR_OUTPUT
   //    "Timer ET" : Time;
   //    "Ouput WORD" : Bool;
   // END_VAR
BEGIN
END_DATA_BLOCK

DATA_BLOCK "DriveConfirmation_Function_Axis 5"   // DB49
VERSION : 0.1
// stored: AutoNumber true, InstanceOfName DriveConfirmation_Function, InstanceOfType FB
"DriveConfirmation_Function"
   // VAR_INPUT
   //    "System RUN" : Bool;
   //    "Drive Ouput Q" : Bool;
   //    "Drive Ready Signal" : Bool;
   //    DelayTime : Time;
   // END_VAR
   // VAR_OUTPUT
   //    "Timer ET" : Time;
   //    "Ouput WORD" : Bool;
   // END_VAR
BEGIN
END_DATA_BLOCK

DATA_BLOCK "DriveConfirmation_Function_Axis1"   // DB45
VERSION : 0.1
// stored: AutoNumber true, InstanceOfName DriveConfirmation_Function, InstanceOfType FB
"DriveConfirmation_Function"
   // VAR_INPUT
   //    "System RUN" : Bool;
   //    "Drive Ouput Q" : Bool;
   //    "Drive Ready Signal" : Bool;
   //    DelayTime : Time;
   // END_VAR
   // VAR_OUTPUT
   //    "Timer ET" : Time;
   //    "Ouput WORD" : Bool;
   // END_VAR
BEGIN
END_DATA_BLOCK

DATA_BLOCK "DriveConfirmation_Function_Axis2"   // DB46
VERSION : 0.1
// stored: AutoNumber true, InstanceOfName DriveConfirmation_Function, InstanceOfType FB
"DriveConfirmation_Function"
   // VAR_INPUT
   //    "System RUN" : Bool;
   //    "Drive Ouput Q" : Bool;
   //    "Drive Ready Signal" : Bool;
   //    DelayTime : Time;
   // END_VAR
   // VAR_OUTPUT
   //    "Timer ET" : Time;
   //    "Ouput WORD" : Bool;
   // END_VAR
BEGIN
END_DATA_BLOCK

DATA_BLOCK "ESB_Buzzer_Block"   // DB33
VERSION : 0.1
// stored: AutoNumber true, InstanceOfName ESB_Flash_Warning_Block, InstanceOfType FB
"ESB_Flash_Warning_Block"
BEGIN
END_DATA_BLOCK

DATA_BLOCK "Ouput_Function_1_Drive1"   // DB4
VERSION : 0.1
// stored: AutoNumber true, InstanceOfName Ouput_Function_1, InstanceOfType FB
"Ouput_Function_1"
BEGIN
END_DATA_BLOCK

DATA_BLOCK "Ouput_Function_1_Drive2"   // DB8
VERSION : 0.1
// stored: AutoNumber true, InstanceOfName Ouput_Function_1, InstanceOfType FB
"Ouput_Function_1"
BEGIN
END_DATA_BLOCK

DATA_BLOCK "Ouput_Function_1_Drive3"   // DB12
VERSION : 0.1
// stored: AutoNumber true, InstanceOfName Ouput_Function_1, InstanceOfType FB
"Ouput_Function_1"
BEGIN
END_DATA_BLOCK

DATA_BLOCK "Ouput_Function_1_Drive4"   // DB17
VERSION : 0.1
// stored: AutoNumber true, InstanceOfName Ouput_Function_1, InstanceOfType FB
"Ouput_Function_1"
BEGIN
END_DATA_BLOCK

DATA_BLOCK "Ouput_Function_1_Drive5"   // DB18
VERSION : 0.1
// stored: AutoNumber true, InstanceOfName Ouput_Function_1, InstanceOfType FB
"Ouput_Function_1"
BEGIN
END_DATA_BLOCK

DATA_BLOCK "Ouput_Function_1_Valve1"   // DB19
VERSION : 0.1
// stored: AutoNumber true, InstanceOfName Ouput_Function_1, InstanceOfType FB
"Ouput_Function_1"
BEGIN
END_DATA_BLOCK

DATA_BLOCK "Ouput_Function_1_Valve3"   // DB26
VERSION : 0.1
// stored: AutoNumber true, InstanceOfName Ouput_Function_1, InstanceOfType FB
"Ouput_Function_1"
BEGIN
END_DATA_BLOCK

DATA_BLOCK "Ouput_Function_1_Valve5"   // DB28
VERSION : 0.1
// stored: AutoNumber true, InstanceOfName Ouput_Function_1, InstanceOfType FB
"Ouput_Function_1"
BEGIN
END_DATA_BLOCK

DATA_BLOCK "MC_Jog_OB1"   // DB56
VERSION : 0.1
// stored: AutoNumber true, InstanceOfName MC_Jog, InstanceOfType FB
"MC_Jog"
BEGIN
END_DATA_BLOCK

DATA_BLOCK "MC_Move_Prog.1"   // DB54
VERSION : 0.1
// stored: AutoNumber true, InstanceOfName MC_Move, InstanceOfType FB
"MC_Move"
BEGIN
END_DATA_BLOCK

DATA_BLOCK "BlowOffTimerCyclic"   // DB84
// stored: AutoNumber true, InstanceOfName TON_SFB, OfSystemLibElement TON, OfSystemLibVersion 1.0
"TON_SFB"
   // VAR_INPUT
   //    IN : Bool;
   //    PT : Time;
   // END_VAR
   // VAR_OUTPUT
   //    Q : Bool;
   //    ET : Time;
   // END_VAR
   // VAR RETAIN
   //    STATE : Byte;
   //    STIME : Time;
   //    ATIME : Time;
   // END_VAR
BEGIN
END_DATA_BLOCK

DATA_BLOCK "Delayed_Message_Function_Timer"   // DB35
// stored: AutoNumber true, InstanceOfName TON_SFB, OfSystemLibElement TON, OfSystemLibVersion 1.0
"TON_SFB"
   // VAR_INPUT
   //    IN : Bool;
   //    PT : Time;
   // END_VAR
   // VAR_OUTPUT
   //    Q : Bool;
   //    ET : Time;
   // END_VAR
   // VAR RETAIN
   //    STATE : Byte;
   //    STIME : Time;
   //    ATIME : Time;
   // END_VAR
BEGIN
END_DATA_BLOCK

DATA_BLOCK "IEC_Timer_0_DB"   // DB31
// stored: AutoNumber true, InstanceOfName TON_SFB, OfSystemLibElement TON, OfSystemLibVersion 1.0
"TON_SFB"
   // VAR_INPUT
   //    IN : Bool;
   //    PT : Time;
   // END_VAR
   // VAR_OUTPUT
   //    Q : Bool;
   //    ET : Time;
   // END_VAR
   // VAR RETAIN
   //    STATE : Byte;
   //    STIME : Time;
   //    ATIME : Time;
   // END_VAR
BEGIN
END_DATA_BLOCK

DATA_BLOCK "IEC_Timer_0_DB_1"   // DB60
// stored: AutoNumber true, InstanceOfName TOF_SFB, OfSystemLibElement TOF, OfSystemLibVersion 1.0
"TOF_SFB"
   // VAR_INPUT
   //    IN : Bool;
   //    PT : Time;
   // END_VAR
   // VAR_OUTPUT
   //    Q : Bool;
   //    ET : Time;
   // END_VAR
   // VAR RETAIN
   //    STATE : Byte;
   //    STIME : Time;
   //    ATIME : Time;
   // END_VAR
BEGIN
END_DATA_BLOCK

DATA_BLOCK "IEC_Timer_0_DB_8"   // DB9
// stored: AutoNumber true, InstanceOfName TON_SFB, OfSystemLibElement TON, OfSystemLibVersion 1.0
"TON_SFB"
   // VAR_INPUT
   //    IN : Bool;
   //    PT : Time;
   // END_VAR
   // VAR_OUTPUT
   //    Q : Bool;
   //    ET : Time;
   // END_VAR
   // VAR RETAIN
   //    STATE : Byte;
   //    STIME : Time;
   //    ATIME : Time;
   // END_VAR
BEGIN
END_DATA_BLOCK

DATA_BLOCK "Move2Done"   // DB88
// stored: AutoNumber true, InstanceOfName TON_SFB, OfSystemLibElement TON, OfSystemLibVersion 1.0
"TON_SFB"
   // VAR_INPUT
   //    IN : Bool;
   //    PT : Time;
   // END_VAR
   // VAR_OUTPUT
   //    Q : Bool;
   //    ET : Time;
   // END_VAR
   // VAR RETAIN
   //    STATE : Byte;
   //    STIME : Time;
   //    ATIME : Time;
   // END_VAR
BEGIN
END_DATA_BLOCK

DATA_BLOCK "RestAferReferenceRun"   // DB52
// stored: AutoNumber true, InstanceOfName TON_SFB, OfSystemLibElement TON, OfSystemLibVersion 1.0
"TON_SFB"
   // VAR_INPUT
   //    IN : Bool;
   //    PT : Time;
   // END_VAR
   // VAR_OUTPUT
   //    Q : Bool;
   //    ET : Time;
   // END_VAR
   // VAR RETAIN
   //    STATE : Byte;
   //    STIME : Time;
   //    ATIME : Time;
   // END_VAR
BEGIN
END_DATA_BLOCK

DATA_BLOCK "Timer_Aanvoerband"   // DB7
// stored: AutoNumber true, InstanceOfName TON_SFB, OfSystemLibElement TON, OfSystemLibVersion 1.0
"TON_SFB"
   // VAR_INPUT
   //    IN : Bool;
   //    PT : Time;
   // END_VAR
   // VAR_OUTPUT
   //    Q : Bool;
   //    ET : Time;
   // END_VAR
   // VAR RETAIN
   //    STATE : Byte;
   //    STIME : Time;
   //    ATIME : Time;
   // END_VAR
BEGIN
END_DATA_BLOCK

DATA_BLOCK "Timer_Retourband_Off"   // DB72
// stored: AutoNumber true, InstanceOfName TOF_SFB, OfSystemLibElement TOF, OfSystemLibVersion 1.0
"TOF_SFB"
   // VAR_INPUT
   //    IN : Bool;
   //    PT : Time;
   // END_VAR
   // VAR_OUTPUT
   //    Q : Bool;
   //    ET : Time;
   // END_VAR
   // VAR RETAIN
   //    STATE : Byte;
   //    STIME : Time;
   //    ATIME : Time;
   // END_VAR
BEGIN
END_DATA_BLOCK

DATA_BLOCK "Timer_Signal_1"   // DB36
// stored: AutoNumber true, InstanceOfName TP_SFB, OfSystemLibElement TP, OfSystemLibVersion 1.0
"TP_SFB"
   // VAR_INPUT
   //    IN : Bool;
   //    PT : Time;
   // END_VAR
   // VAR_OUTPUT
   //    Q : Bool;
   //    ET : Time;
   // END_VAR
   // VAR RETAIN
   //    STATE : Byte;
   //    STIME : Time;
   //    ATIME : Time;
   // END_VAR
BEGIN
END_DATA_BLOCK

DATA_BLOCK "Timer_Trilgoten"   // DB5
// stored: AutoNumber true, InstanceOfName TON_SFB, OfSystemLibElement TON, OfSystemLibVersion 1.0
"TON_SFB"
   // VAR_INPUT
   //    IN : Bool;
   //    PT : Time;
   // END_VAR
   // VAR_OUTPUT
   //    Q : Bool;
   //    ET : Time;
   // END_VAR
   // VAR RETAIN
   //    STATE : Byte;
   //    STIME : Time;
   //    ATIME : Time;
   // END_VAR
BEGIN
END_DATA_BLOCK

DATA_BLOCK "TotalProductsCounter"   // DB22
// stored: AutoNumber true, InstanceOfName CTU_SFB, OfSystemLibElement CTU, OfSystemLibVersion 1.0
"CTU_SFB"
   // VAR_INPUT
   //    CU : Bool;
   //    R : Bool;
   //    PV : Int;
   // END_VAR
   // VAR_OUTPUT
   //    Q : Bool;
   //    CV : Int;
   // END_VAR
   // VAR RETAIN
   //    CUO : Bool;
   // END_VAR
BEGIN
END_DATA_BLOCK

DATA_BLOCK "Uitlooptimer_Aanvoerband"   // DB10
// stored: AutoNumber true, InstanceOfName TON_SFB, OfSystemLibElement TON, OfSystemLibVersion 1.0
"TON_SFB"
   // VAR_INPUT
   //    IN : Bool;
   //    PT : Time;
   // END_VAR
   // VAR_OUTPUT
   //    Q : Bool;
   //    ET : Time;
   // END_VAR
   // VAR RETAIN
   //    STATE : Byte;
   //    STIME : Time;
   //    ATIME : Time;
   // END_VAR
BEGIN
END_DATA_BLOCK

DATA_BLOCK "Uitlooptimer_Trilgoten"   // DB11
// stored: AutoNumber true, InstanceOfName TON_SFB, OfSystemLibElement TON, OfSystemLibVersion 1.0
"TON_SFB"
   // VAR_INPUT
   //    IN : Bool;
   //    PT : Time;
   // END_VAR
   // VAR_OUTPUT
   //    Q : Bool;
   //    ET : Time;
   // END_VAR
   // VAR RETAIN
   //    STATE : Byte;
   //    STIME : Time;
   //    ATIME : Time;
   // END_VAR
BEGIN
END_DATA_BLOCK

DATA_BLOCK "WalsOff_delay"   // DB13
// stored: AutoNumber true, InstanceOfName TON_SFB, OfSystemLibElement TON, OfSystemLibVersion 1.0
"TON_SFB"
   // VAR_INPUT
   //    IN : Bool;
   //    PT : Time;
   // END_VAR
   // VAR_OUTPUT
   //    Q : Bool;
   //    ET : Time;
   // END_VAR
   // VAR RETAIN
   //    STATE : Byte;
   //    STIME : Time;
   //    ATIME : Time;
   // END_VAR
BEGIN
END_DATA_BLOCK

DATA_BLOCK "WarningTimer2"   // DB32
// stored: AutoNumber true, InstanceOfName TON_SFB, OfSystemLibElement TON, OfSystemLibVersion 1.0
"TON_SFB"
   // VAR_INPUT
   //    IN : Bool;
   //    PT : Time;
   // END_VAR
   // VAR_OUTPUT
   //    Q : Bool;
   //    ET : Time;
   // END_VAR
   // VAR RETAIN
   //    STATE : Byte;
   //    STIME : Time;
   //    ATIME : Time;
   // END_VAR
BEGIN
END_DATA_BLOCK

DATA_BLOCK "ProductBuffer_V3_DB"   // DB90
VERSION : 0.1
// stored: AutoNumber true, InstanceOfName ProductBuffer_V3, InstanceOfType FB
"ProductBuffer_V3"
BEGIN
END_DATA_BLOCK
